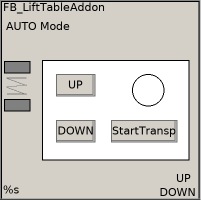
VISUALIZATION V_LiftTableAddon  // 201x200
VAR_IN_OUT
	{attribute 'VAR_IN_OUT_AS_POINTER'}
	fbFunction 		: FB_LiftTableAddon;
	fbEmuFunction	: FB_LiftTableAddonEmulation;
END_VAR
    Rectangle (0,0 200x200), colour toggle: fbFunction.HW_Outputs.LiftDown OR fbFunction.HW_Outputs.LiftUp
    Rectangle (0,180 200x20), "%s", text variable: fbFunction.ConfigFunction.FunctionName
    Label (0,0 200x15), "FB_LiftTableAddon"
    Label (166,172 35x13), "UP", invisible if: NOT fbFunction.HW_Outputs.LiftUp
    Label (155,185 45x15), "DOWN", invisible if: NOT fbFunction.HW_Outputs.LiftDown
    Polyline (26,78) (7,78) (26,85) (7,87) (26,94) (7,94), colour toggle: fbFunction.HW_Outputs.LiftUp OR fbFunction.HW_Outputs.LiftDown
    Rectangle (4,99 26x12), tooltip "Lower lift sensor", colour toggle: fbFunction.HW_Inputs.Lift.SensorPosDown
    Rectangle (4,61 26x12), tooltip "Upper lift sensor", colour toggle: fbFunction.HW_Inputs.Lift.SensorPosUp
    RoundedRectangle (42,60 147x100)
    Button (56,120 39x22), "DOWN"
        tap fbEmuFunction.DebugOpDown
    Button (111,120 66x22), "StartTransp"
        tap fbEmuFunction.DebugOpStartTransp
    Ellipse (132,74 32x32), colour toggle: fbFunction.HW_Outputs.StartTransport
    Button (56,74 39x22), "UP"
        tap fbEmuFunction.DebugOpUp
    Label (3,20 79x13), "AUTO Mode", invisible if: fbFunction.Settings.OperatorPanelEnable
END_VISUALIZATION

(* stored: Version 1.1.0.1, ProductVersion 3.1.4024.9
   Visu V_LiftTableAddon: Id {e2f4520e-0ec6-492c-9376-13d4069da813} *)
